TYPE TMPType :
(
	TMPType_Default := 0 //常规分子泵
)UINT;
END_TYPE

(* stored: Version 1.1.0.1, ProductVersion 3.1.4024.4
   DUT TMPType: Id {d485b005-34b4-4b1c-8391-35857a1245dc} *)
